(*
SPDX-FileCopyrightText: Â© 2026 Oleksandr Tiutyk <trofimich@gmail.com>
SPDX-License-Identifier: MIT
License: https://opensource.org/license/mit
*)

(*!
<summary>Represents a child automation component whose simulation override can be configured.</summary>
*)

INTERFACE IChildConfigurableSimulatable EXTENDS IChildSimulatable

(*!
<summary>Configures the simulation mode override setting for this child component.</summary>
<param name="value">Override setting (INHERITED, ON, or OFF).</param>
*)
METHOD SetSimulationModeOverride
VAR_INPUT
	value : SIMULATION_MODE_OVERRIDE;
END_VAR
END_METHOD

END_INTERFACE

(* stored: Version 1.1.0.1
   Itf IChildConfigurableSimulatable: Id {7067e270-a72e-4b40-a559-79b7dea6079f}
   Method SetSimulationModeOverride: Id {b0ed9d3c-7f83-40a4-b58c-915e8a072ecc} *)
